Staubli VAL3: refreshStatic.pgx

program refreshStatic()
  local num l_nLocal
  local string l_sMessage
begin
  //
  // CREATE THE LIST
  // define your list size for default
  //
  cls()
  call use:setSizeList(19,0,19,11)
  call use:setView(bLarge)
  //
  switch nViewMode
    case 0
      call use:listcreate(" OUT ")
    break
    case 1
      call use:listcreate(" IN ")
    break
    case 2
      call use:listcreate("COUNT")
    break
  endSwitch
  //

end
